(* CoDeSys 2.3 export: FB_BLOCK.EXP *)

(* POU FB_Block, ST *)
(*Variables in inputs so that they can be written from outside*)
FUNCTION_BLOCK FB_Block
VAR_INPUT
	StrValue : STRING;
	Data : ST_StandardTypes;
END_VAR
VAR_OUTPUT
END_VAR
VAR
END_VAR
;
END_FUNCTION_BLOCK
